// SIMATIC S7-200 project (STEP 7-Micro/WIN), CPU 221 REL 01.10

SYMBOL_TABLE USER1
MODE             I0.0
ON_              I0.1
OFF_             I0.2
ON_CT1           M0.0
ON_CT2           M0.1
DEN1             Q0.0
DEN2             Q0.1
DEN              Q0.2
END_SYMBOL_TABLE

ORGANIZATION_BLOCK MAIN:OB1
TITLE=PROGRAM COMMENTS
BEGIN
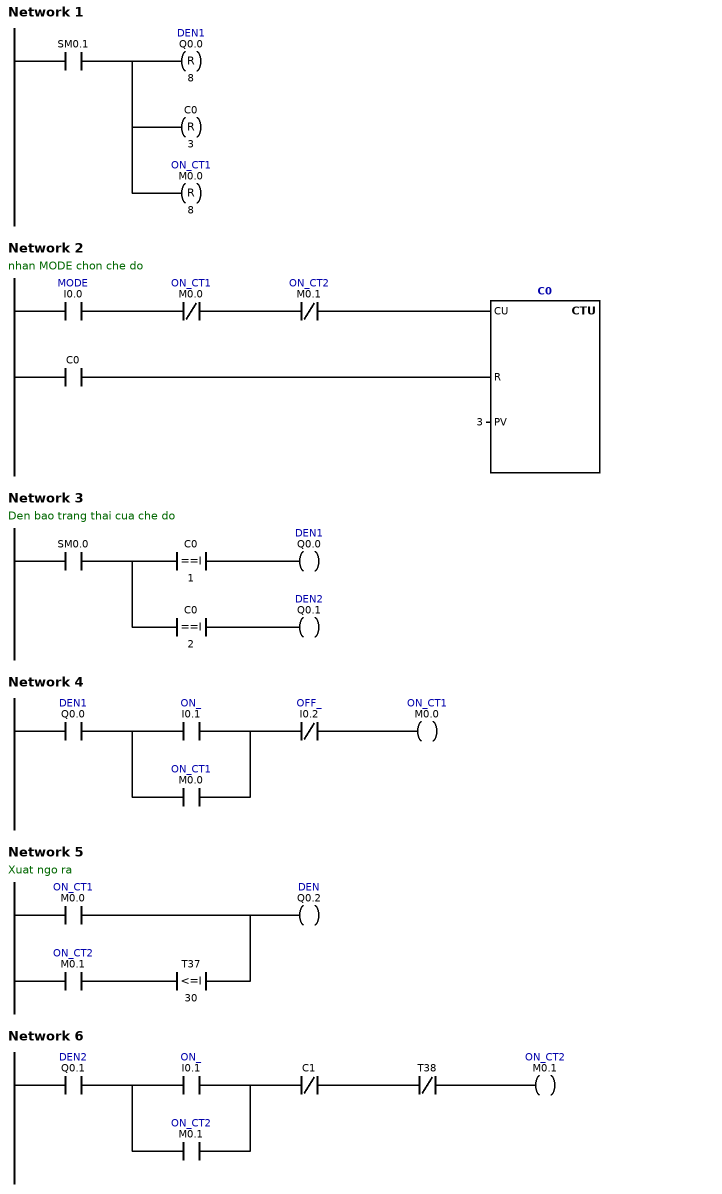
Network 1
LD     SM0.1
R      DEN1:Q0.0, 8
R      C0, 3
R      ON_CT1:M0.0, 8
Network 2
// nhan MODE chon che do
LD     MODE:I0.0
AN     ON_CT1:M0.0
AN     ON_CT2:M0.1
LD     C0
CTU    C0, 3
Network 3
// Den bao trang thai cua che do
LD     SM0.0
LPS
AW=    C0, 1
=      DEN1:Q0.0
LPP
AW=    C0, 2
=      DEN2:Q0.1
Network 4
LD     DEN1:Q0.0
LD     ON_:I0.1
O      ON_CT1:M0.0
ALD
AN     OFF_:I0.2
=      ON_CT1:M0.0
Network 5
// Xuat ngo ra
LD     ON_CT1:M0.0
LD     ON_CT2:M0.1
AW<=   T37, 30
OLD
=      DEN:Q0.2
Network 6
LD     DEN2:Q0.1
LD     ON_:I0.1
O      ON_CT2:M0.1
ALD
AN     C1
AN     T38
=      ON_CT2:M0.1
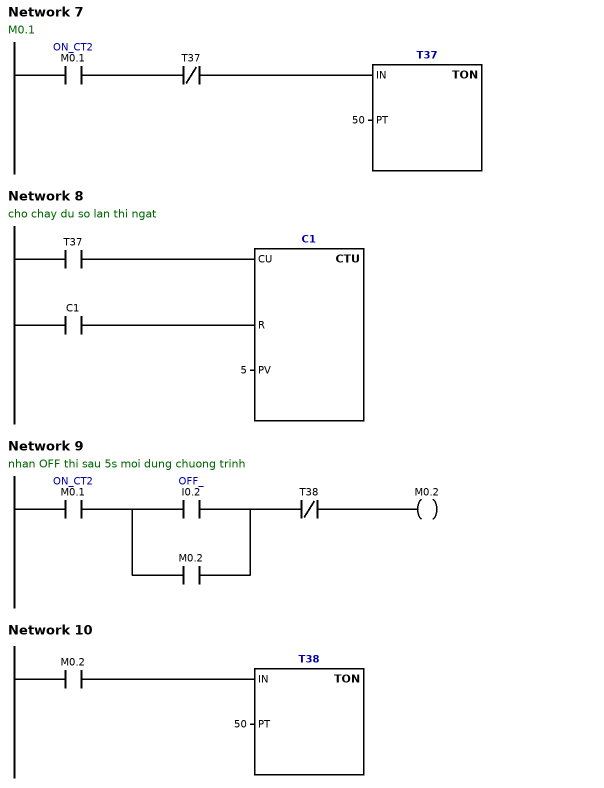
Network 7
// M0.1
LD     ON_CT2:M0.1
AN     T37
TON    T37, 50
Network 8
// cho chay du so lan thi ngat
LD     T37
LD     C1
CTU    C1, 5
Network 9
// nhan OFF thi sau 5s moi dung chuong trinh
LD     ON_CT2:M0.1
LD     OFF_:I0.2
O      M0.2
ALD
AN     T38
=      M0.2
Network 10
LD     M0.2
TON    T38, 50
END_ORGANIZATION_BLOCK
